Fanuc KAREL source: kt00271.KL

PROGRAM KT00271
%NOLOCKGROUP
VAR
H1 : ARRAY[2] OF SHORT
I2:INTEGER
OUT:BOOLEAN
BEGIN
H1[1]=2
I2=3
OUT=(H1[1]=I2)
END KT00271
